FUNCTION_BLOCK FB_System_WP_Ablaufsteuerung
VAR_IN_OUT
	Zustand				: ST_System_WP_Zustand;
	Stellwert			: ST_System_WP_Stellwert;
	Steuerung			: ST_System_WP_Steuerung;
END_VAR
VAR_INPUT
	Zustand_SV_KW			: ST_SV_Zustand;
	Zustand_SV_WW			: ST_SV_Zustand;
	Zustand_WP				: ST_WP_Zustand;
END_VAR
VAR_OUTPUT
END_VAR
VAR
END_VAR

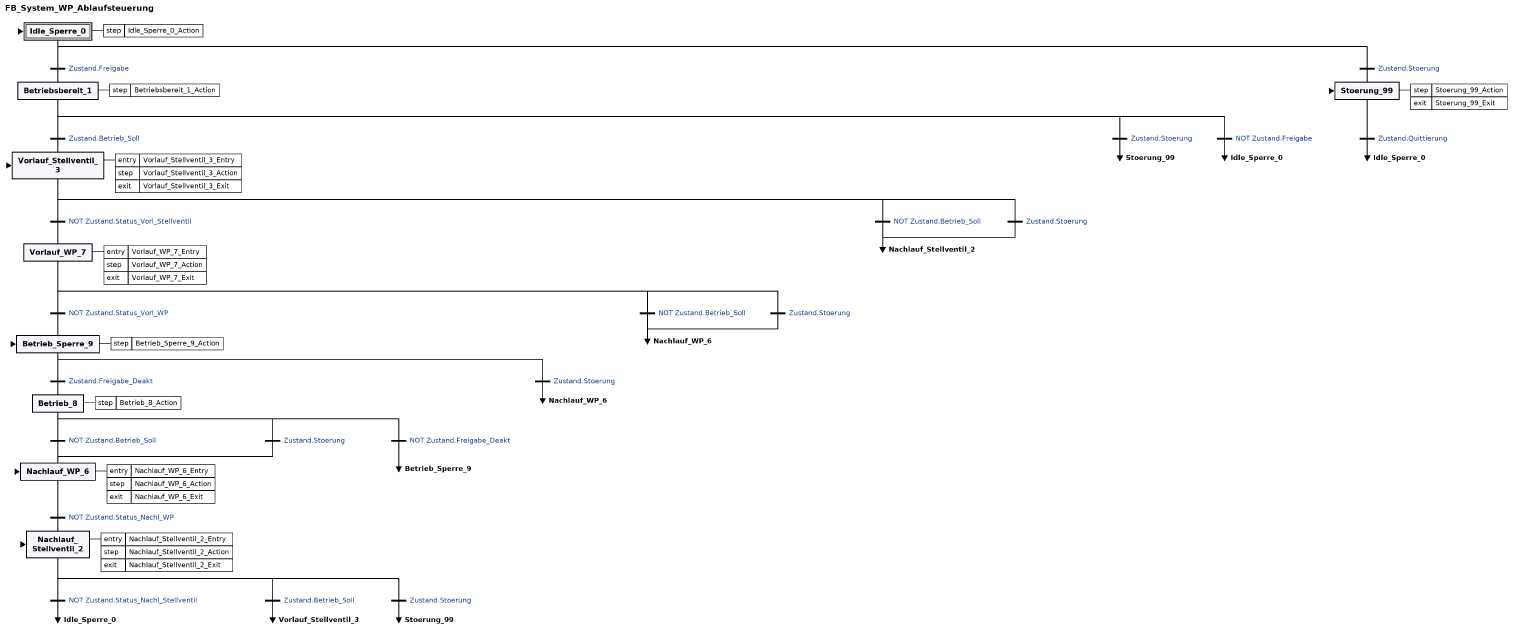
INITIAL_STEP Idle_Sperre_0:
    Idle_Sperre_0_Action(N);  // step action
END_STEP
TRANSITION FROM Idle_Sperre_0 TO Betriebsbereit_1
    := Zustand.Freigabe;
END_TRANSITION
TRANSITION FROM Idle_Sperre_0 TO Stoerung_99
    := Zustand.Stoerung;
END_TRANSITION
STEP Stoerung_99:
    Stoerung_99_Action(N);  // step action
    Stoerung_99_Exit(P0);  // exit action
END_STEP
TRANSITION FROM Stoerung_99 TO Idle_Sperre_0
    := Zustand.Quittierung;
END_TRANSITION
STEP Betriebsbereit_1:
    Betriebsbereit_1_Action(N);  // step action
END_STEP
TRANSITION FROM Betriebsbereit_1 TO Vorlauf_Stellventil_3
    := Zustand.Betrieb_Soll;
END_TRANSITION
TRANSITION FROM Betriebsbereit_1 TO Stoerung_99
    := Zustand.Stoerung;
END_TRANSITION
TRANSITION FROM Betriebsbereit_1 TO Idle_Sperre_0
    := NOT Zustand.Freigabe;
END_TRANSITION
STEP Vorlauf_Stellventil_3:
    Vorlauf_Stellventil_3_Entry(P1);  // entry action
    Vorlauf_Stellventil_3_Action(N);  // step action
    Vorlauf_Stellventil_3_Exit(P0);  // exit action
END_STEP
TRANSITION FROM Vorlauf_Stellventil_3 TO Vorlauf_WP_7
    := NOT Zustand.Status_Vorl_Stellventil;
END_TRANSITION
TRANSITION FROM Vorlauf_Stellventil_3 TO Nachlauf_Stellventil_2
    := NOT Zustand.Betrieb_Soll;
END_TRANSITION
TRANSITION FROM Vorlauf_Stellventil_3 TO Nachlauf_Stellventil_2
    := Zustand.Stoerung;
END_TRANSITION
STEP Vorlauf_WP_7:
    Vorlauf_WP_7_Entry(P1);  // entry action
    Vorlauf_WP_7_Action(N);  // step action
    Vorlauf_WP_7_Exit(P0);  // exit action
END_STEP
TRANSITION FROM Vorlauf_WP_7 TO Betrieb_Sperre_9
    := NOT Zustand.Status_Vorl_WP;
END_TRANSITION
TRANSITION FROM Vorlauf_WP_7 TO Nachlauf_WP_6
    := NOT Zustand.Betrieb_Soll;
END_TRANSITION
TRANSITION FROM Vorlauf_WP_7 TO Nachlauf_WP_6
    := Zustand.Stoerung;
END_TRANSITION
STEP Betrieb_Sperre_9:
    Betrieb_Sperre_9_Action(N);  // step action
END_STEP
TRANSITION FROM Betrieb_Sperre_9 TO Betrieb_8
    := Zustand.Freigabe_Deakt;
END_TRANSITION
TRANSITION FROM Betrieb_Sperre_9 TO Nachlauf_WP_6
    := Zustand.Stoerung;
END_TRANSITION
STEP Betrieb_8:
    Betrieb_8_Action(N);  // step action
END_STEP
TRANSITION FROM Betrieb_8 TO Nachlauf_WP_6
    := NOT Zustand.Betrieb_Soll;
END_TRANSITION
TRANSITION FROM Betrieb_8 TO Nachlauf_WP_6
    := Zustand.Stoerung;
END_TRANSITION
TRANSITION FROM Betrieb_8 TO Betrieb_Sperre_9
    := NOT Zustand.Freigabe_Deakt;
END_TRANSITION
STEP Nachlauf_WP_6:
    Nachlauf_WP_6_Entry(P1);  // entry action
    Nachlauf_WP_6_Action(N);  // step action
    Nachlauf_WP_6_Exit(P0);  // exit action
END_STEP
TRANSITION FROM Nachlauf_WP_6 TO Nachlauf_Stellventil_2
    := NOT Zustand.Status_Nachl_WP;
END_TRANSITION
STEP Nachlauf_Stellventil_2:
    Nachlauf_Stellventil_2_Entry(P1);  // entry action
    Nachlauf_Stellventil_2_Action(N);  // step action
    Nachlauf_Stellventil_2_Exit(P0);  // exit action
END_STEP
TRANSITION FROM Nachlauf_Stellventil_2 TO Idle_Sperre_0
    := NOT Zustand.Status_Nachl_Stellventil;
END_TRANSITION
TRANSITION FROM Nachlauf_Stellventil_2 TO Vorlauf_Stellventil_3
    := Zustand.Betrieb_Soll;
END_TRANSITION
TRANSITION FROM Nachlauf_Stellventil_2 TO Stoerung_99
    := Zustand.Stoerung;
END_TRANSITION

ACTION Betrieb_8_Action:
(* Stellwert setzen *)
Stellwert.Anford_SV_KW	:= TRUE;
Stellwert.Anford_SV_WW	:= TRUE;
Stellwert.Anford_WP		:= TRUE;

(* Zustand setzen *)
Zustand.Status				:= E_System_WP_Zustand_Status_Betrieb;
END_ACTION

ACTION Betrieb_Sperre_9_Action:
(* Stellwert setzen *)
Stellwert.Anford_SV_KW	:= TRUE;
Stellwert.Anford_SV_WW	:= TRUE;
Stellwert.Anford_WP		:= TRUE;

(* Zustand setzen *)
Zustand.Status				:= E_System_WP_Zustand_Status_Betrieb_Sperre;
END_ACTION

ACTION Betriebsbereit_1_Action:
(* Stellwert setzen *)
Stellwert.Anford_SV_KW	:= FALSE;
Stellwert.Anford_SV_WW	:= FALSE;
Stellwert.Anford_WP		:= FALSE;

(* Zustand setzen *)
Zustand.Status			:= E_System_BWK_Zustand_Status_Betriebsbereit;
END_ACTION

ACTION Idle_Sperre_0_Action:
(* Stellwert setzen *)
Stellwert.Anford_SV_KW	:= FALSE;
Stellwert.Anford_SV_WW	:= FALSE;
Stellwert.Anford_WP		:= FALSE;

(* Zustand setzen *)
Zustand.Status			:= E_System_BWK_Zustand_Status_Idle_Sperre;


(* Quittierungszustand auf False setzen, damit das System bei einer erneuten Störung nicht direkt wieder angeschaltet wird *)
Steuerung.Quittierung	:= FALSE;
END_ACTION

ACTION Nachlauf_Stellventil_2_Action:
(* Stellwert setzen *)
Stellwert.Anford_SV_KW	:= FALSE;
Stellwert.Anford_SV_WW	:= FALSE;
Stellwert.Anford_WP		:= FALSE;

(* Zustand setzen *)
Zustand.Status				:= E_System_WP_Zustand_Status_Nachl_Stellventil;
Zustand.Status_Nachl_SV_KW	:= Zustand_SV_KW.Stellung OR Zustand_SV_KW.Stellungwechsel10;
Zustand.Status_Nachl_SV_WW	:= Zustand_SV_WW.Stellung OR Zustand_SV_WW.Stellungwechsel10;
END_ACTION

ACTION Nachlauf_Stellventil_2_Entry:
Zustand.Status_Nachl_Stellventil	:= TRUE;
END_ACTION

ACTION Nachlauf_Stellventil_2_Exit:
Zustand.Status_Nachl_Stellventil	:= FALSE;
END_ACTION

ACTION Nachlauf_WP_6_Action:
(* Stellwert setzen *)
Stellwert.Anford_SV_KW	:= TRUE;
Stellwert.Anford_SV_WW	:= TRUE;
Stellwert.Anford_WP		:= FALSE;

(* Zustand setzen *)
Zustand.Status				:= E_System_WP_Zustand_Status_Nachl_WP;
Zustand.Status_Nachl_WP		:= Zustand_WP.Betrieb OR Zustand_WP.Status_Nachl;
END_ACTION

ACTION Nachlauf_WP_6_Entry:
Zustand.Status_Nachl_WP		:= TRUE;
END_ACTION

ACTION Nachlauf_WP_6_Exit:
Zustand.Status_Nachl_WP		:= FALSE;
END_ACTION

ACTION Stoerung_99_Action:
(* Stellwert setzen *)
Stellwert.Anford_SV_KW	:= FALSE;
Stellwert.Anford_SV_WW	:= FALSE;
Stellwert.Anford_WP		:= FALSE;

(* Zustand setzen *)
Zustand.Stoerung			:= TRUE;
Zustand.Status			:= E_System_WP_Zustand_Status_Stoerung;
END_ACTION

ACTION Stoerung_99_Exit:
Zustand.Stoerung	:= FALSE;
END_ACTION

ACTION Vorlauf_Stellventil_3_Action:
(* Stellwert setzen *)
Stellwert.Anford_SV_KW	:= TRUE;
Stellwert.Anford_SV_WW	:= TRUE;
Stellwert.Anford_WP		:= FALSE;

(* Zustand setzen *)
Zustand.Status				:= E_System_WP_Zustand_Status_Vorl_Stellventil;
Zustand.Status_Vorl_SV_KW	:= NOT(Zustand_SV_WW.Stellung AND NOT Zustand_SV_WW.Stellungwechsel01);
Zustand.Status_Vorl_SV_WW	:= NOT(Zustand_SV_KW.Stellung AND NOT Zustand_SV_KW.Stellungwechsel01);
END_ACTION

ACTION Vorlauf_Stellventil_3_Entry:
Zustand.Status_Vorl_Stellventil	:= TRUE;
END_ACTION

ACTION Vorlauf_Stellventil_3_Exit:
Zustand.Status_Vorl_Stellventil	:= FALSE;
END_ACTION

ACTION Vorlauf_WP_7_Action:
(* Stellwert setzen *)
Stellwert.Anford_SV_KW	:= TRUE;
Stellwert.Anford_SV_WW	:= TRUE;
Stellwert.Anford_WP		:= TRUE;

(* Zustand setzen *)
Zustand.Status				:= E_System_WP_Zustand_Status_Vorl_WP;
Zustand.Status_Vorl_WP		:= NOT(Zustand_WP.Betrieb AND NOT Zustand_WP.Status_Vorl);
END_ACTION

ACTION Vorlauf_WP_7_Entry:
Zustand.Status_Vorl_WP		:= TRUE;
END_ACTION

ACTION Vorlauf_WP_7_Exit:
Zustand.Status_Vorl_WP		:= FALSE;
END_ACTION

END_FUNCTION_BLOCK

(* stored: Version 1.1.0.1, ProductVersion 3.1.4024.9
   POU FB_System_WP_Ablaufsteuerung: Id {3bf07550-6197-4aee-8df4-acb5e67ed09c}, SpecialFunc None
   Action Betrieb_8_Action: Id {6d7f2233-8279-4c7c-8e36-16e2a067fb04}
   Action Betrieb_Sperre_9_Action: Id {834867e7-d026-45a7-b69f-98198ae0a9ca}
   Action Betriebsbereit_1_Action: Id {6df923c5-bc1a-42e2-aadf-8bba9d0a8151}
   Action Idle_Sperre_0_Action: Id {5c412867-7f58-4ccd-8c42-4f14d3ddbfc3}
   Action Nachlauf_Stellventil_2_Action: Id {d90ae415-2fec-44a9-ae8b-e6d0d5525489}
   Action Nachlauf_Stellventil_2_Entry: Id {36b58db0-4064-409b-8565-d26b46fcb69b}
   Action Nachlauf_Stellventil_2_Exit: Id {f83b0f60-c387-44bf-b5b7-8cc1fc05c3b9}
   Action Nachlauf_WP_6_Action: Id {f51be516-6c32-4bc8-90aa-5e69098daeb1}
   Action Nachlauf_WP_6_Entry: Id {a4f84ffd-4829-4f35-9d7c-c7f3f7712f0d}
   Action Nachlauf_WP_6_Exit: Id {c47266d5-8dba-478a-aa9d-4b7bbe2ffeb6}
   Action Stoerung_99_Action: Id {33bfc1ee-5233-4611-abef-a250db91d50a}
   Action Stoerung_99_Exit: Id {b698068c-7f9b-441e-93f5-643e9ddeba42}
   Action Vorlauf_Stellventil_3_Action: Id {34901f28-8c04-4ce5-9d88-36de6bece2c1}
   Action Vorlauf_Stellventil_3_Entry: Id {312cfde3-ba5c-4c2b-b24a-08153eb57ca6}
   Action Vorlauf_Stellventil_3_Exit: Id {3543e07e-e28e-4dfe-bbaf-e36fd41ae203}
   Action Vorlauf_WP_7_Action: Id {7aa854a4-516f-4f34-b79f-14a90f6146cd}
   Action Vorlauf_WP_7_Entry: Id {0a0ad522-2440-414b-923d-6bb4a19f92a3}
   Action Vorlauf_WP_7_Exit: Id {acce0fe4-6813-4e7f-af6e-59d81c5a3c2c} *)
